// TIA Portal V16 export
// export: Created 2024-09-05T17:39:18.4082604Z, ExportSetting WithDefaults, DisplayName Totally Integrated Automation Portal, DisplayVersion V16 Update 6, DisplayName TIA Portal Version Control Interface, DisplayVersion V16 Update 2, DisplayName TIA Portal Openness, DisplayVersion V16 Update 6, DisplayName STEP 7 Professional, DisplayVersion V16 Update 6, DisplayName STEP 7 Safety, DisplayVersion V16, DisplayName WinCC Advanced, DisplayVersion V16 Update 6
DATA_BLOCK "St1Insertion"   // DB15
{ S7_Optimized_Access := 'TRUE' }
VERSION : 0.1
// stored: AutoNumber true, DBAccessibleFromOPCUA true, IsOnlyStoredInLoadMemory false, IsRetainMemResEnabled false, IsWriteProtectedInAS false, MemoryReserve 100
   VAR
      ExpectedSensors : Array[0..20] of Bool;
      UsedSensors : Array[0..20] of Bool;
      SensorsState : Array[0..20] of Bool;
      SensorsNOK : Array[0..20] of Bool;
      NOKList : Array[0..20] of Int;
      InsertionOK : Bool := TRUE;
      InsertionNOK : Bool := FALSE;
      InsertionEmpty : Bool := TRUE;
      EmptyBits : Array[0..20] of Bool;
      FullBits : Array[0..20] of Bool;
   END_VAR
BEGIN
   ExpectedSensors[0..20] := FALSE;
   UsedSensors[0..20] := FALSE;
   SensorsState[0..20] := FALSE;
   SensorsNOK[0..20] := FALSE;
   NOKList[0..20] := 0;
   EmptyBits[0..20] := FALSE;
   FullBits[0] := FALSE;
   FullBits[1..17] := TRUE;
   FullBits[18..20] := FALSE;
END_DATA_BLOCK
